// SIMATIC S7-200 project (STEP 7-Micro/WIN), CPU 221 REL 01.10

ORGANIZATION_BLOCK MAIN:OB1
TITLE=PROGRAM COMMENTS
BEGIN
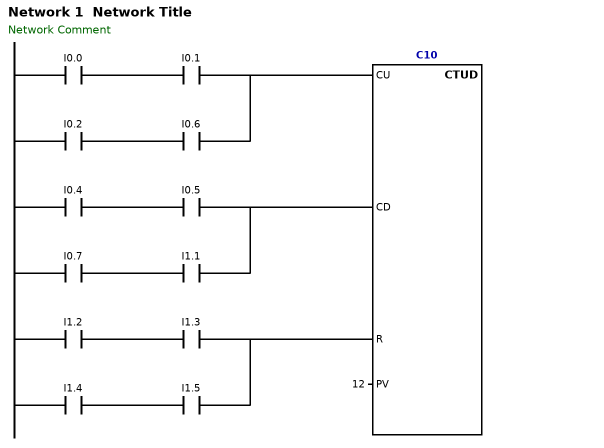
Network 1 // Network Title
// Network Comment
LD     I0.0
A      I0.1
LD     I0.2
A      I0.6
OLD
LD     I0.4
A      I0.5
LD     I0.7
A      I1.1
OLD
LD     I1.2
A      I1.3
LD     I1.4
A      I1.5
OLD
CTUD   C10, 12
END_ORGANIZATION_BLOCK
